FUNCTION_BLOCK AB_TO_AQ (* Converts an AB (BYTE) adapter to an AQ (Quarter Byte) adapter *)
  (* Standard: 61499-2; Description: Copyright (c) 2026 Meisterschulen am Ostbahnhof SPDX-License-Identifier: EPL-2.0 *)
  (* Version 1.0, 2026-05-16, Franz Höpfinger, Meisterschulen am Ostbahnhof, Initial Version *)
  PACKAGE adapter::conversion::unidirectional;
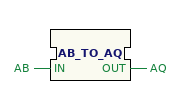
  SOCKETS
    IN : adapter::types::unidirectional::AB; (* BYTE Input *)
  END_SOCKETS
  PLUGS
    OUT : adapter::types::unidirectional::AQ; (* AQ Output *)
  END_PLUGS
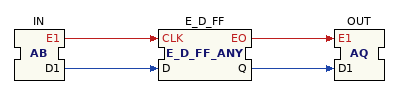
  FBS
    E_D_FF : iec61499::events::E_D_FF_ANY;
  END_FBS
  EVENT_CONNECTIONS
    IN.E1 TO E_D_FF.CLK;
    E_D_FF.EO TO OUT.E1;
  END_CONNECTIONS
  DATA_CONNECTIONS
    IN.D1 TO E_D_FF.D;
    E_D_FF.Q TO OUT.D1;
  END_CONNECTIONS
END_FUNCTION_BLOCK
